// TIA Portal project "Bandas_Cajas" (V17)
// Vorlageprojekt für das Buch mit Zielsystem S7-1200

(* hardware
DEVICE "S7-1200-Station_1"  S7-1200 Station
   slot 0: "Baugruppenträger_0"  Rack  V1.0
   slot 1: "PLC_1"  CPU 1214C DC/DC/DC  6ES7 214-1AG40-0XB0  V4.1
*)

// ===== PLC "PLC_1"  CPU 1214C DC/DC/DC =====

VAR_GLOBAL   // PLC tag table "Standard-Variablentabelle"
   "Start" AT %E0.0 : Bool;
   "Stop" AT %E0.1 : Bool;
   "Reset" AT %I0.2 : Bool;
   "Belt_2" AT %Q0.1 : Bool;
   "Start_light" AT %Q0.2 : Bool;
   "Belt_1" AT %Q0.0 : Bool;
   "Stop_light" AT %Q0.3 : Bool;
   "Emitter" AT %Q0.4 : Bool;
   "Sensor_Caja" AT %I0.4 : Bool;
   "Conteo_Cajas" AT %QW30 : Int;
END_VAR

// folder: System blocks/Program resources

DATA_BLOCK "Cantidad_Cajas"   // DB1
{ S7_Optimized_Access := 'TRUE' }
AUTHOR : Simatic
FAMILY : IEC
NAME : CNTR
VERSION : 1.0
// stored: InstanceOfName IEC_COUNTER
"IEC_COUNTER"
BEGIN
END_DATA_BLOCK

// folder: (top level)

FUNCTION "MHJ-PLC-Lab-Function-S71200" : Void   // FC9000, SCL
{ S7_Optimized_Access := 'TRUE' }
VERSION : 0.1
   VAR_TEMP
      rdTimeReturn : Int;
      outputTime : DTL;
      SyncVal : Byte;
      forVal : Int;
      forVal_2 : Int;
      Value : Byte;
   END_VAR
   VAR CONSTANT
      CompVal : Byte := 16#34;
      Value_01 : Byte := 16#11;
      Value_01_DW : DWord := 16#A165_D992;
      Value_02_DW : DWord := 16#58BE_4401;
   END_VAR
BEGIN

   #Value:=PEEK(area := 16#82,
        dbNumber := 0,
        byteOffset := 511);
   #Value := #Value + 1;

   POKE(area := 16#82,
        dbNumber := 0,
        byteOffset := 511,
        value := #Value);

   POKE(area:=16#81,
        dbNumber:=0,
        byteOffset:=1016,
        value:=#Value_01_DW);
   POKE(area := 16#81,
        dbNumber := 0,
        byteOffset := 1020,
        value := #Value_02_DW);

   POKE(area := 16#81,
        dbNumber := 0,
        byteOffset := 511,
        value := B#16#00);

   FOR #forVal := 0 TO 120 DO
       FOR #forVal_2:=0 TO 10 DO
           #rdTimeReturn:=RD_SYS_T(#outputTime);
           #rdTimeReturn := WR_SYS_T(#outputTime);
           #rdTimeReturn := RD_SYS_T(#outputTime);
           #rdTimeReturn := WR_SYS_T(#outputTime);
       END_FOR;
       #SyncVal:= PEEK(area := 16#81,
                      dbNumber := 0,
                      byteOffset := 511);
       IF #SyncVal = #CompVal THEN
          GOTO M_1;
       END_IF;
   END_FOR;
   RETURN;

   M_1:
   POKE(area := 16#81,
        dbNumber := 0,
        byteOffset := 511,
        value := B#16#0);
END_FUNCTION

ORGANIZATION_BLOCK "Main"   // OB1, LAD, ProgramCycle
TITLE = "Main Program Sweep (Cycle)"
{ S7_Optimized_Access := 'TRUE' }
VERSION : 0.1
   VAR_INPUT
      Initial_Call : Bool;   // Initial call of this OB
      Remanence : Bool;   // =True, if remanent data are available
   END_VAR
   VAR_TEMP   // added for the SCL form of the ladder/FBD networks
      _w1 : Bool;
   END_VAR
BEGIN

REGION Network 1: Konnektierungsbaustein für PLC-Lab
   // Im Netzwerk 1 wird der Konnektierungsbaustein für PLC-Lab aufgerufen.
   // Dieser Aufruf darf nicht entfernt werden!
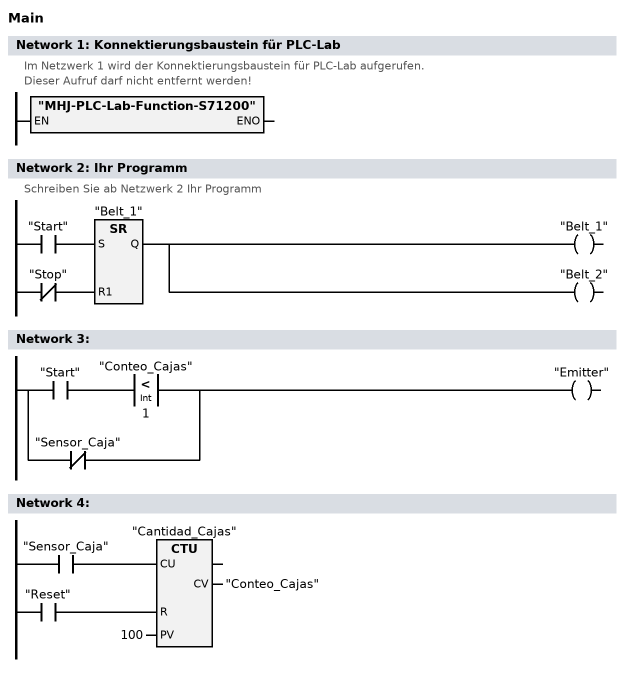
   RUNG wire#powerrail
      "MHJ-PLC-Lab-Function-S71200"()
   END_RUNG
   // the same network as SCL:
   "MHJ-PLC-Lab-Function-S71200"();
END_REGION

REGION Network 2: Ihr Programm
   // Schreiben Sie ab Netzwerk 2 Ihr Programm
   RUNG wire#powerrail
      Contact( "Start" )
      S_SR(operand := "Belt_1", r1 := wire#w1)
      wire#w2
      Coil( "Belt_1" )
   END_RUNG
   RUNG wire#powerrail
      I_Contact( "Stop" )
   END_RUNG wire#w1
   RUNG wire#w2
      Coil( "Belt_2" )
   END_RUNG
   // the same network as SCL:
   IF "Start" THEN
       "Belt_1" := TRUE;   // SR flip-flop
   END_IF;
   IF NOT "Stop" THEN "Belt_1" := FALSE; END_IF;
   #_w1 := "Belt_1";
   "Belt_1" := "Belt_1";
   "Belt_2" := #_w1;
END_REGION

REGION Network 3
   RUNG wire#powerrail
      Contact( "Start" )
      { S7_Templates := "SrcType := Int" } LT_Contact(in1 := "Conteo_Cajas", in2 := 1)
      wire#w1
      Coil( "Emitter" )
   END_RUNG
   RUNG wire#powerrail
      I_Contact( "Sensor_Caja" )
   END_RUNG wire#w1
   // the same network as SCL:
   "Emitter" := ("Start" AND ("Conteo_Cajas" < 1)) OR NOT "Sensor_Caja";
END_REGION

REGION Network 4
   "Cantidad_Cajas".CTU(CU := "Sensor_Caja", R := "Reset", PV := 100, CV => "Conteo_Cajas");
END_REGION
END_ORGANIZATION_BLOCK